RoboDK station: kr30 cnc 041619 2.rdk

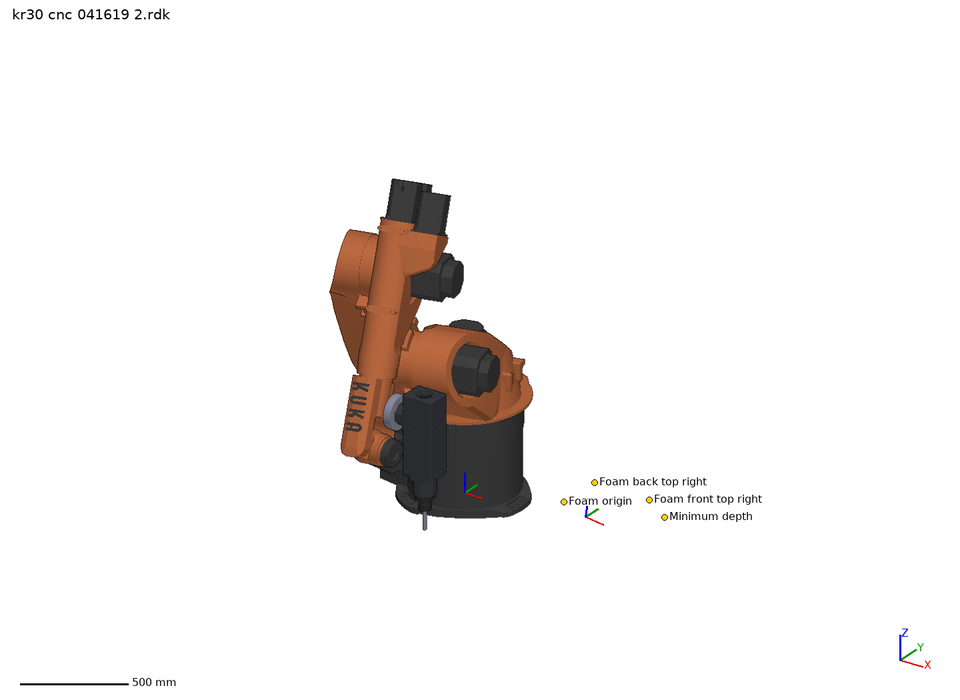
[picture v0: the station drawn from its stored meshes, robots at their saved joint values, targets as dots, program paths as lines]
Station kr30 cnc 041619 2. Poses are relative to the parent item; angles as X-Y-Z fixed-axis rotations.
  - frame KUKA KR 30 HA Base at (0, 0, 0) mm
    - robot KUKA KR 30 HA: 6 axes, payload 30 kg, reach 2033 mm, repeatability 0.05 mm, weight 665 kg
        modified DH rows (alpha deg, a mm, theta deg, d mm): 0, 0, 0, 815; -90, 350, 0, 0; 0, 850, -90, 0; -90, 145, 0, 820; 90, 0, 0, 0; -90, 0, 180, 170
        joint limits [-185, -135, -120, -350, -119, -350] to [185, 35, 158, 350, 119, 350]; home [0, -90, 90, 0, 0, 0]; saved at [75.216, -55.782, 118.463, 76.804, -83.275, -26.54]
      - tool 1/2" End Mill TCP, TCP at (337.71, -2.2, 160.57) mm, size 692.9 x 170 x 256 mm
    - target Foam origin (Cartesian target) at (1070.87, -730.54, 545.36) mm, rotated rx -134.27 ry 89.31 rz 136.22 deg; joints [20.571, -65.631, 133.307, -70.576, -81.708, 21.487] of KUKA KR 30 HA
    - target Foam back top right (Cartesian target) at (1070.87, -482.98, 545.36) mm, rotated rx -134.27 ry 89.31 rz 136.22 deg; joints [8.23, -68.302, 138.029, -81.988, -86.539, 20.562] of KUKA KR 30 HA
    - target Foam front top right (Cartesian target) at (1372.4, -476.64, 537.69) mm, rotated rx -134.27 ry 89.31 rz 136.21 deg; joints [6.181, -54.802, 114.144, -84.508, -86.194, 30.998] of KUKA KR 30 HA
    - target Minimum depth (Cartesian target) at (1405.34, -397.62, 426.66) mm, rotated rx -134.27 ry 89.31 rz 136.21 deg; joints [2.841, -47.623, 111.899, -87.216, -88.124, 26.187] of KUKA KR 30 HA
  - frame Milling Reference at (-4814.43, -552.71, 1443.13) mm
    - object TABLE HEIGHT NOT YET SET at (7007.1, -1218.12, -920.21) mm, size 1193.8 x 965.2 x 609.6 mm, geometry from welding_table.sld
  - machining project RhinoPart Settings: C:/Users/Julian Ramirez.DESKTOP-JVDE542/Desktop/ELMER SHEET 1 TEST 3.nc | rotZ(0) | rotX(0)*rotY(0) | rotz(0)*rotY(270)
  - object box at (500, 500, 500) mm, size 250 x 250 x 250 mm, geometry from box.sld
  - frame Frame 3 at (1029.96, -496.81, 362.28) mm, rotated rx 0 ry 8.45 rz 0 deg
    - object RhinoPart at (0, 0, 0) mm
